FUNCTION_BLOCK ControlModule (* Composite Function Block Type *)
  (* Standard: 61499-2 *)
  (* Version 0.0, 2011-12-28, 4DIAC-IDE, 4DIAC-Consortium *)
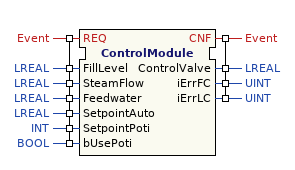
  EVENT_INPUT
    REQ WITH FillLevel, SteamFlow, Feedwater, SetpointAuto, SetpointPoti, bUsePoti; (* Normal Execution Request *)
  END_EVENT
  EVENT_OUTPUT
    CNF WITH ControlValve, iErrFC, iErrLC; (* Execution Confirmation *)
  END_EVENT
  VAR_INPUT
    FillLevel : LREAL; (* Input event qualifier *)
    SteamFlow : LREAL;
    Feedwater : LREAL;
    SetpointAuto : LREAL;
    SetpointPoti : INT;
    bUsePoti : BOOL;
  END_VAR
  VAR_OUTPUT
    ControlValve : LREAL; (* Output event qualifier *)
    iErrFC : UINT;
    iErrLC : UINT;
  END_VAR
  FBS
    FlowController : FlowController;
    LevelController : LevelController;
    ControlComputation : ControlComputation;
  END_FBS
  EVENT_CONNECTIONS
    REQ TO LevelController.REQ;
    FlowController.CNF TO CNF;
    LevelController.CNF TO ControlComputation.REQ;
    ControlComputation.CNF TO FlowController.REQ;
  END_CONNECTIONS
  DATA_CONNECTIONS
    FillLevel TO LevelController.Measurement;
    SetpointAuto TO LevelController.SetpointExt;
    SetpointPoti TO LevelController.SetpointPoti;
    bUsePoti TO LevelController.bUsePoti;
    FlowController.ControlOut TO ControlValve;
    FlowController.iErr TO iErrFC;
    LevelController.iErr TO iErrLC;
    LevelController.ControlOut TO ControlComputation.Input1;
    ControlComputation.ControlOut TO FlowController.Setpoint;
    Feedwater TO ControlComputation.Input2;
    SteamFlow TO ControlComputation.Input3;
  END_CONNECTIONS
END_FUNCTION_BLOCK
